(* Logix 5000 project; controller Drives_Line1 1756-L72 rev 20.13; software revision 20.04; part 2 of 21 *)
(* tags used below, declared in another part *)
   TofStitch_Z2 : TIMER;
   TofStitch_Z3 : TIMER;
   TofWatchDogMaster : TIMER;
   _bv_tmp : INT;
   Bridle_01 : UDT_Bridle_3M;
   Bridle_01_FB_Diff : REAL;
   Bridle_01_FB_Update_Valid : BOOL;
   Bridle_01b_FBCounts_mm : REAL;
   Bridle_02 : UDT_Bridle_2M;
   Bridle_03 : UDT_Bridle_2M;
   Bridle_04 : UDT_Bridle_3M;
   cu : UDT_Pinchroll;
   Entry_Accu : UDT_Entry_Accu;
   EntryCmd : UDT_Commands_Zone;
   EntryConfig : UDT_Config_Zone;
   EntryCtrl : UDT_Control_Zone;
   EntryFdbks : UDT_Feedbacks_Zone;
   EntrySetpoints : UDT_Setpoints_Zone;
   EntryStat : UDT_Status_Zone;
   Exit_Accu : UDT_Exit_Accu;
   ExitCtrl : UDT_Control_Zone;
   ExitStat : UDT_Status_Zone;
   In_Commands : UDT_Commands;
   In_Config : UDT_Config;
   In_Setpoints : UDT_Setpoints;
   LineCmd : UDT_Commands_Line;
   LineConfig : UDT_Config_Line;
   LineCtrl : UDT_Control_Line;
   LineFdbks : UDT_Feedbacks_Line;
   LineSetpoints : UDT_Setpoints_Line;
   LineStat : UDT_Status_Line;
   nbrstiychout : DINT;
   Out_Feedbacks : UDT_Fdbks;
   Out_Status : UDT_Status;
   Pinchroll_1 : UDT_Pinchroll;
   Pinchroll_2 : UDT_Pinchroll;
   TestConfig_Line : UDT_Config_Line;
   Unwinder_1 : UDT_Unwinder;
   Unwinder_2 : UDT_Unwinder;
   voirmw : BOOL;
   zConfigFromMaster : BOOL;
   zSimulation : BOOL;
(* P00_Line, continued *)

ROUTINE R12_Line_State   (* ladder *)
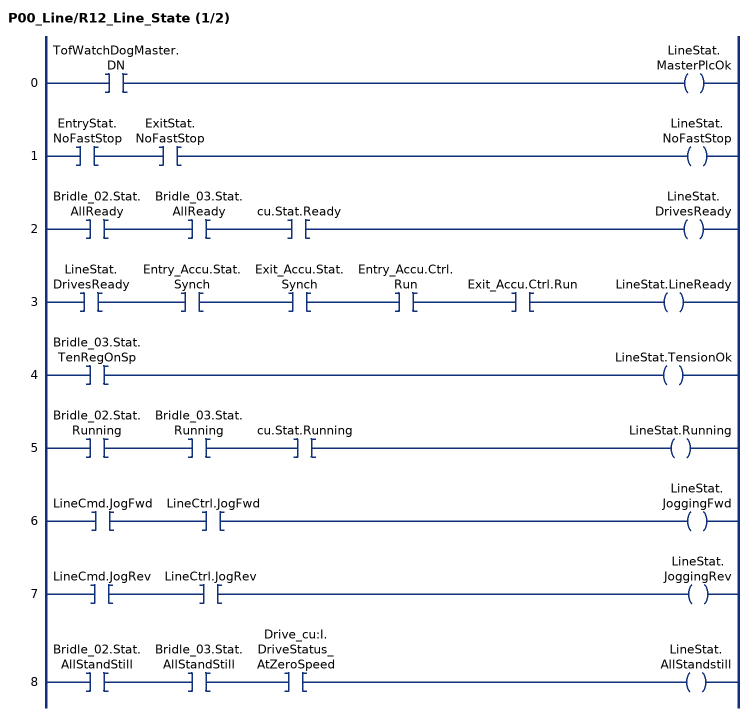
   0: XIC(TofWatchDogMaster.DN)OTE(LineStat.MasterPlcOk);
   1: XIC(EntryStat.NoFastStop)XIC(ExitStat.NoFastStop)OTE(LineStat.NoFastStop);
   2: XIC(Bridle_02.Stat.AllReady)XIC(Bridle_03.Stat.AllReady)XIC(cu.Stat.Ready)OTE(LineStat.DrivesReady);
   3: XIC(LineStat.DrivesReady)XIC(Entry_Accu.Stat.Synch)XIC(Exit_Accu.Stat.Synch)XIC(Entry_Accu.Ctrl.Run)XIC(Exit_Accu.Ctrl.Run)OTE(LineStat.LineReady);
   4: XIC(Bridle_03.Stat.TenRegOnSp)OTE(LineStat.TensionOk);
   5: XIC(Bridle_02.Stat.Running)XIC(Bridle_03.Stat.Running)XIC(cu.Stat.Running)OTE(LineStat.Running);
   6: XIC(LineCmd.JogFwd)XIC(LineCtrl.JogFwd)OTE(LineStat.JoggingFwd);
   7: XIC(LineCmd.JogRev)XIC(LineCtrl.JogRev)OTE(LineStat.JoggingRev);
   8: XIC(Bridle_02.Stat.AllStandStill)XIC(Bridle_03.Stat.AllStandStill)XIC(Drive_cu:I.DriveStatus_AtZeroSpeed)OTE(LineStat.AllStandstill);
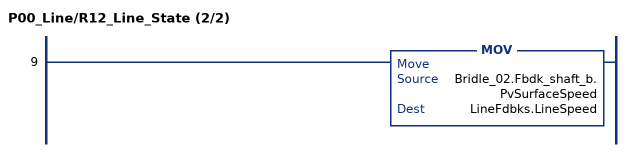
   9: MOV(Bridle_02.Fbdk_shaft_b.PvSurfaceSpeed,LineFdbks.LineSpeed);
END_ROUTINE

ROUTINE R13_Line_Control   (* ladder *)
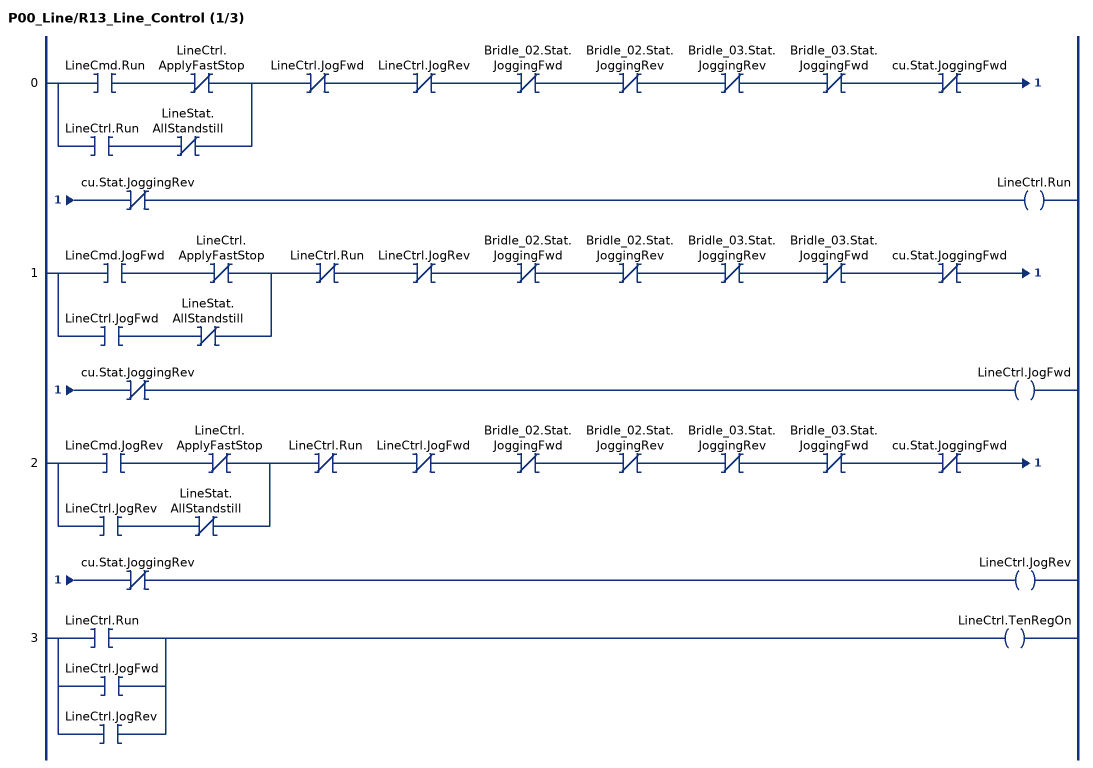
   0: [XIC(LineCmd.Run) XIO(LineCtrl.ApplyFastStop) ,XIC(LineCtrl.Run) XIO(LineStat.AllStandstill) ]XIO(LineCtrl.JogFwd)XIO(LineCtrl.JogRev)XIO(Bridle_02.Stat.JoggingFwd)XIO(Bridle_02.Stat.JoggingRev)XIO(Bridle_03.Stat.JoggingRev)XIO(Bridle_03.Stat.JoggingFwd)XIO(cu.Stat.JoggingFwd)XIO(cu.Stat.JoggingRev)OTE(LineCtrl.Run);
   1: [XIC(LineCmd.JogFwd) XIO(LineCtrl.ApplyFastStop) ,XIC(LineCtrl.JogFwd) XIO(LineStat.AllStandstill) ]XIO(LineCtrl.Run)XIO(LineCtrl.JogRev)XIO(Bridle_02.Stat.JoggingFwd)XIO(Bridle_02.Stat.JoggingRev)XIO(Bridle_03.Stat.JoggingRev)XIO(Bridle_03.Stat.JoggingFwd)XIO(cu.Stat.JoggingFwd)XIO(cu.Stat.JoggingRev)OTE(LineCtrl.JogFwd);
   2: [XIC(LineCmd.JogRev) XIO(LineCtrl.ApplyFastStop) ,XIC(LineCtrl.JogRev) XIO(LineStat.AllStandstill) ]XIO(LineCtrl.Run)XIO(LineCtrl.JogFwd)XIO(Bridle_02.Stat.JoggingFwd)XIO(Bridle_02.Stat.JoggingRev)XIO(Bridle_03.Stat.JoggingRev)XIO(Bridle_03.Stat.JoggingFwd)XIO(cu.Stat.JoggingFwd)XIO(cu.Stat.JoggingRev)OTE(LineCtrl.JogRev);
   3: [XIC(LineCtrl.Run) ,XIC(LineCtrl.JogFwd) ,XIC(LineCtrl.JogRev) ]OTE(LineCtrl.TenRegOn);
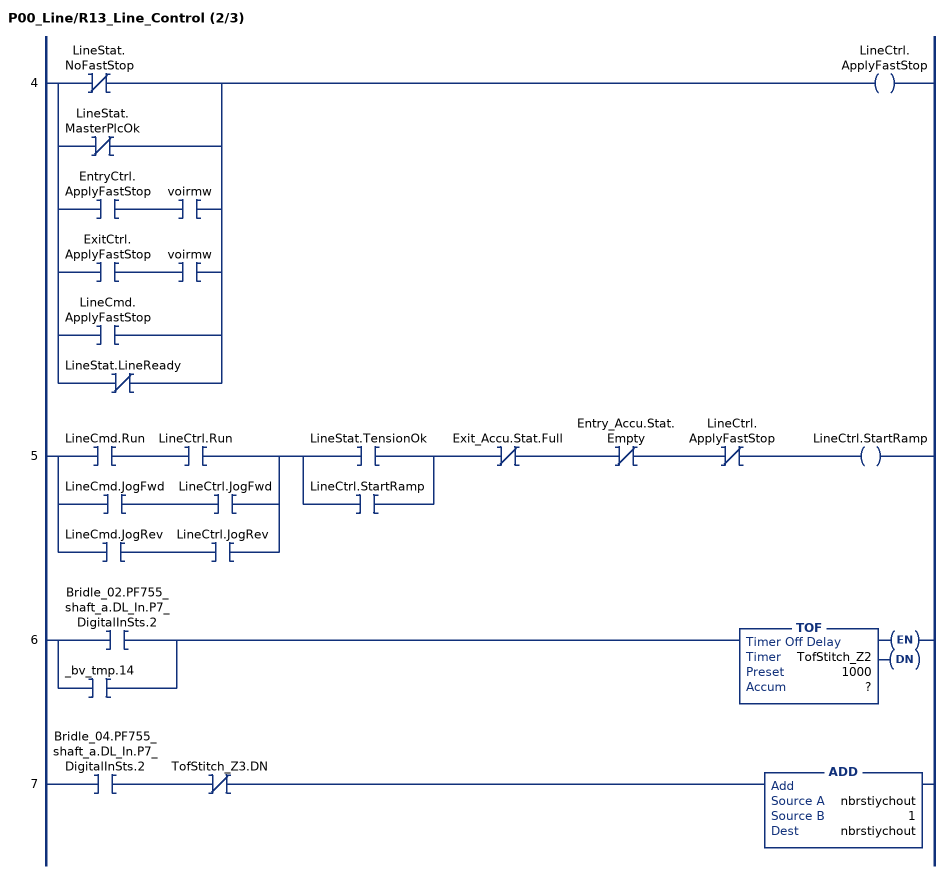
   4: [XIO(LineStat.NoFastStop) ,XIO(LineStat.MasterPlcOk) ,XIC(EntryCtrl.ApplyFastStop) XIC(voirmw) ,XIC(ExitCtrl.ApplyFastStop) XIC(voirmw) ,XIC(LineCmd.ApplyFastStop) ,XIO(LineStat.LineReady) ]OTE(LineCtrl.ApplyFastStop);
   5: [XIC(LineCmd.Run) XIC(LineCtrl.Run) ,XIC(LineCmd.JogFwd) XIC(LineCtrl.JogFwd) ,XIC(LineCmd.JogRev) XIC(LineCtrl.JogRev) ][XIC(LineStat.TensionOk) ,XIC(LineCtrl.StartRamp) ]XIO(Exit_Accu.Stat.Full)XIO(Entry_Accu.Stat.Empty)XIO(LineCtrl.ApplyFastStop)OTE(LineCtrl.StartRamp);
   6: [XIC(Bridle_02.PF755_shaft_a.DL_In.P7_DigitalInSts.2) ,XIC(_bv_tmp.14) ]TOF(TofStitch_Z2,?,?);
   7: XIC(Bridle_04.PF755_shaft_a.DL_In.P7_DigitalInSts.2)XIO(TofStitch_Z3.DN)ADD(nbrstiychout,1,nbrstiychout);
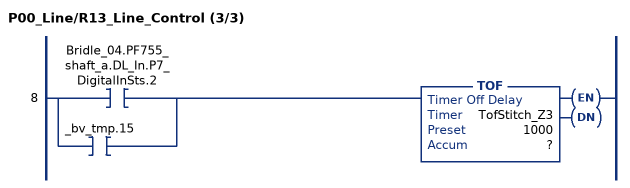
   8: [XIC(Bridle_04.PF755_shaft_a.DL_In.P7_DigitalInSts.2) ,XIC(_bv_tmp.15) ]TOF(TofStitch_Z3,?,?);
END_ROUTINE

ROUTINE R15_Ramp_LineRef_Vp   (* function block diagram *)
   SHEET 1   // Select speed reference
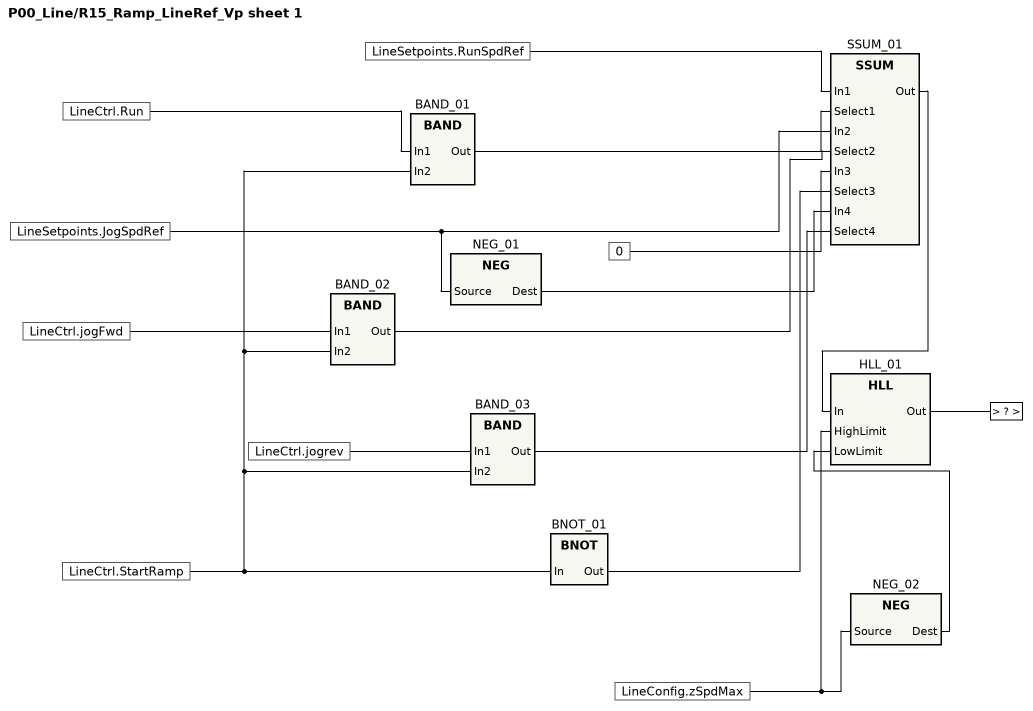
   BAND_02 : BAND(In1 := LineCtrl.jogFwd, In2 := LineCtrl.StartRamp);
   BAND_01 : BAND(In1 := LineCtrl.Run, In2 := LineCtrl.StartRamp);
   NEG_01 : NEG(Source := LineSetpoints.JogSpdRef);
   BAND_03 : BAND(In1 := LineCtrl.jogrev, In2 := LineCtrl.StartRamp);
   BNOT_01 : BNOT(In := LineCtrl.StartRamp);
   SSUM_01 : SSUM(In1 := LineSetpoints.RunSpdRef, Select1 := BAND_01.Out, In2 := LineSetpoints.JogSpdRef, Select2 := BAND_02.Out, In3 := 0, Select3 := BNOT_01.Out, In4 := NEG_01.Dest, Select4 := BAND_03.Out);
   NEG_02 : NEG(Source := LineConfig.zSpdMax);
   HLL_01 : HLL(In := SSUM_01.Out, HighLimit := LineConfig.zSpdMax, LowLimit := NEG_02.Dest);
   WIRE(?) := HLL_01.Out;
   SHEET 2   // Select acceleration rate
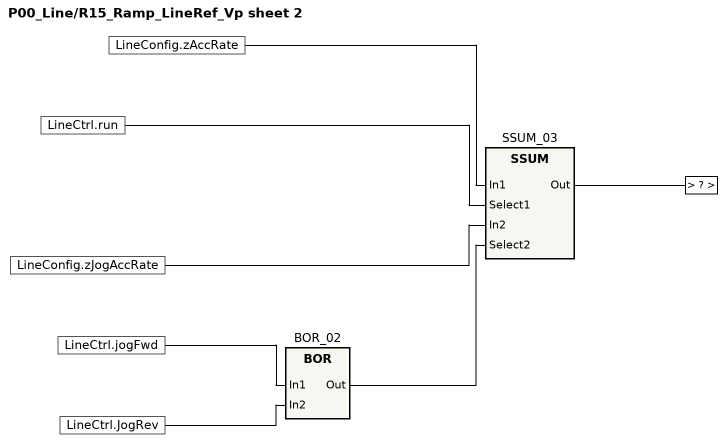
   BOR_02 : BOR(In1 := LineCtrl.jogFwd, In2 := LineCtrl.JogRev);
   SSUM_03 : SSUM(In1 := LineConfig.zAccRate, Select1 := LineCtrl.run, In2 := LineConfig.zJogAccRate, Select2 := BOR_02.Out);
   WIRE(?) := SSUM_03.Out;
   SHEET 3   // Select deceleration rate
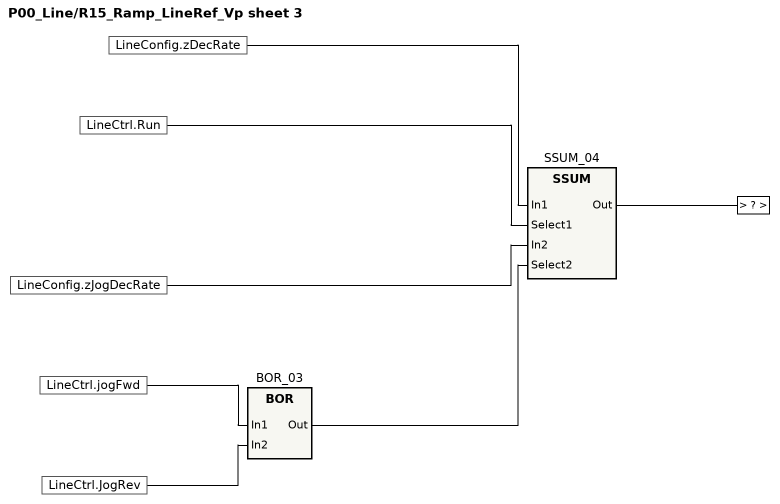
   BOR_03 : BOR(In1 := LineCtrl.jogFwd, In2 := LineCtrl.JogRev);
   SSUM_04 : SSUM(In1 := LineConfig.zDecRate, Select1 := LineCtrl.Run, In2 := LineConfig.zJogDecRate, Select2 := BOR_03.Out);
   WIRE(?) := SSUM_04.Out;
   SHEET 4   // S-Curve line speed (Vp)
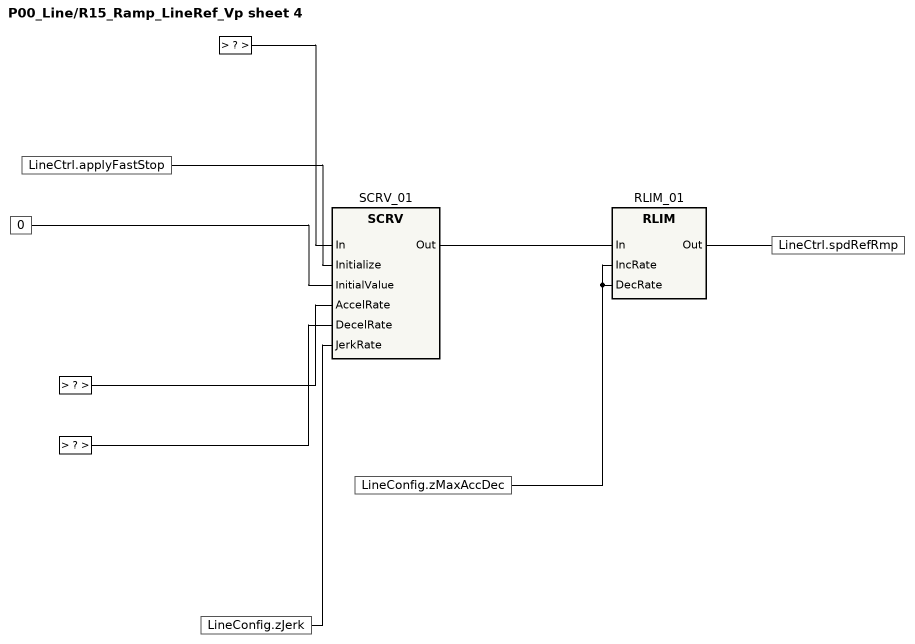
   SCRV_01 : SCRV(In := WIRE(?), Initialize := LineCtrl.applyFastStop, InitialValue := 0, AccelRate := WIRE(?), DecelRate := WIRE(?), JerkRate := LineConfig.zJerk);
   RLIM_01 : RLIM(In := SCRV_01.Out, IncRate := LineConfig.zMaxAccDec, DecRate := LineConfig.zMaxAccDec);
   LineCtrl.spdRefRmp := RLIM_01.Out;
END_ROUTINE

ROUTINE R999_Test   (* ladder *)
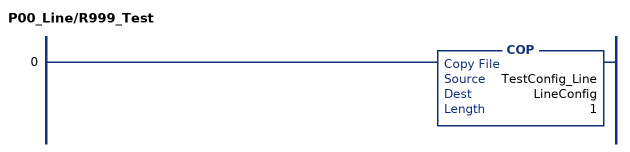
   0: COP(TestConfig_Line,LineConfig,1);
END_ROUTINE

ROUTINE R99_To_Master   (* ladder *)
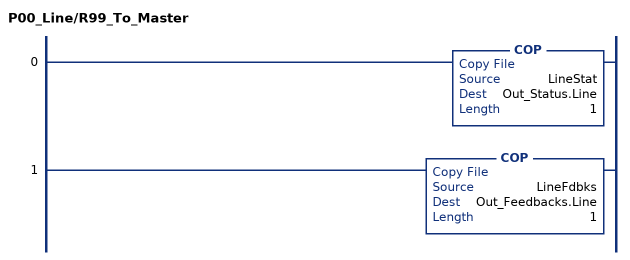
   0: COP(LineStat,Out_Status.Line,1);
   1: COP(LineFdbks,Out_Feedbacks.Line,1);
END_ROUTINE
END_PROGRAM

PROGRAM P01_Entry_Zone   (* main routine R00_Main *)
VAR
   BAND_10 : FBD_BOOLEAN_AND := (In3 := 1, In4 := 1, In5 := 1, In6 := 1, In7 := 1, In8 := 1);
   BAND_11 : FBD_BOOLEAN_AND := (In3 := 1, In4 := 1, In5 := 1, In6 := 1, In7 := 1, In8 := 1);
   BAND_12 : FBD_BOOLEAN_AND := (In3 := 1, In4 := 1, In5 := 1, In6 := 1, In7 := 1, In8 := 1);
   BNOT_01 : FBD_BOOLEAN_NOT := (Out := 1);
   BNOT_04 : FBD_BOOLEAN_NOT := (Out := 1);
   BOR_01 : FBD_BOOLEAN_OR;
   Entry_PosPv_Shear_Stitch : REAL := 2345.455;
   Entry_PosPv_Stitch_HOC : DINT;
   Entry_PosSp_AtShear : DINT := 1650;
   Entry_PosSp_AtStitch_EOC : DINT := 2345;
   Entry_PosSp_AtStitch_HOC : DINT := 1650;
   EOC_PosStitchStep : DINT;
   EOC_ToShearStep : DINT;
   HLL_01 : HL_LIMIT := (HighLimit := 0.5, LowLimit := -0.5);
   HLL_02 : HL_LIMIT := (HighAlarm := 1, LowAlarm := 1, Status := 16#0000_0003, InstructFault := 1, LimitsInv := 1);
   HOC_ToStitchStep : DINT;
   NEG_01 : FBD_MATH_ADVANCED := (Source := 0.5, Dest := -0.5);
   NEG_05 : FBD_MATH_ADVANCED := (Source := 0.1, Dest := -0.1);
   NEG_06 : FBD_MATH_ADVANCED;
   ons : BOOL[32] := ([0] := 1, [1] := 1);
   RLIM_02 : RATE_LIMITER := (IncRate := 0.25, DecRate := 0.25, RTSTime := 1, DeltaT := 0.05);
   SCRV_02 : S_CURVE := (Initialize := 1, RTSTime := 1, DeltaT := 0.05);
   SEL_02 : SELECT := (In1 := 0.08, SelectorIn := 1);
   SSUM_03 : SELECTED_SUMMER := (Gain1 := 1.0, In2 := 0.1, Gain2 := 1.0, In3 := -0.1, Gain3 := 1.0, Gain4 := 1.0, Select4 := 1, Gain5 := 1.0, Gain6 := 1.0, Gain7 := 1.0, Gain8 := 1.0);
   SSUM_06 : SELECTED_SUMMER := (In1 := 0.04, Gain1 := 1.0, In2 := 0.083, Gain2 := 1.0, Gain3 := 1.0, Gain4 := 1.0, Gain5 := 1.0, Gain6 := 1.0, Gain7 := 1.0, Gain8 := 1.0);
   SSUM_08 : SELECTED_SUMMER := (In1 := 0.04, Gain1 := 1.0, In2 := 0.083, Gain2 := 1.0, Gain3 := 1.0, Gain4 := 1.0, Gain5 := 1.0, Gain6 := 1.0, Gain7 := 1.0, Gain8 := 1.0);
   SSUM_09 : SELECTED_SUMMER := (In1 := 0.15, Gain1 := 1.0, In2 := 0.1, Gain2 := 1.0, Gain3 := 1.0, Gain4 := 1.0, Gain5 := 1.0, Gain6 := 1.0, Gain7 := 1.0, Gain8 := 1.0);
   Ton_EOC_Sensor : TIMER := (PRE := 1000, ACC := 1000, EN := 1, DN := 1);
   TonRefOn : TIMER := (PRE := 750);
   zEntry_Dist_Pinch_Shear : REAL := 1650.0;
   zEntry_Dist_ShearToStitch : REAL := 695.0;
   zMaxSpdEntryNotSync : REAL := 0.08;
END_VAR

ROUTINE R00_Main   (* ladder *)
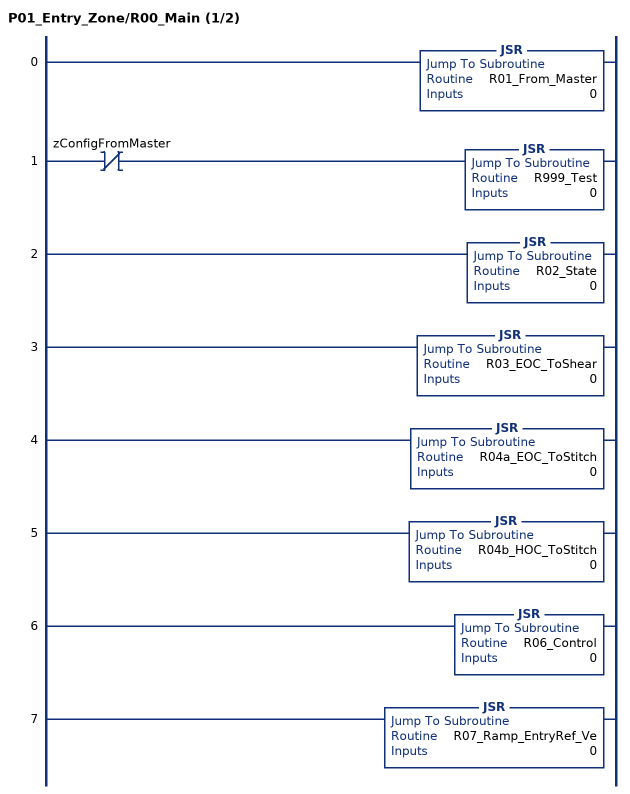
   0: JSR(R01_From_Master,0);
   1: XIO(zConfigFromMaster)JSR(R999_Test,0);
   2: JSR(R02_State,0);
   3: JSR(R03_EOC_ToShear,0);
   4: JSR(R04a_EOC_ToStitch,0);
   5: JSR(R04b_HOC_ToStitch,0);
   6: JSR(R06_Control,0);
   7: JSR(R07_Ramp_EntryRef_Ve,0);
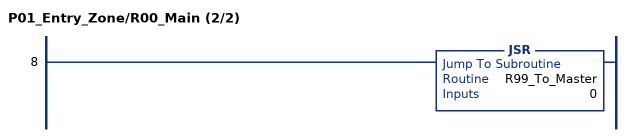
   8: JSR(R99_To_Master,0);
END_ROUTINE

ROUTINE R01_From_Master   (* ladder *)
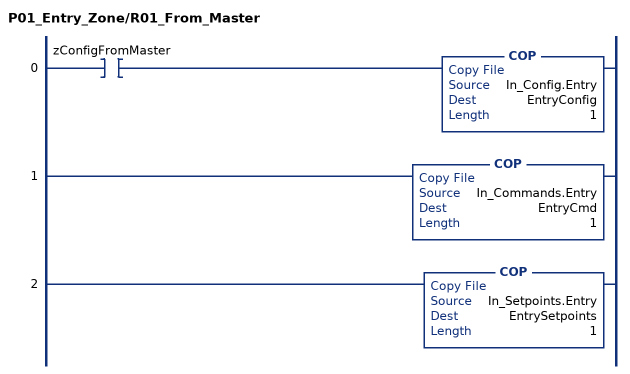
   0: XIC(zConfigFromMaster)COP(In_Config.Entry,EntryConfig,1);
   1: COP(In_Commands.Entry,EntryCmd,1);
   2: COP(In_Setpoints.Entry,EntrySetpoints,1);
END_ROUTINE

ROUTINE R02_State   (* ladder *)
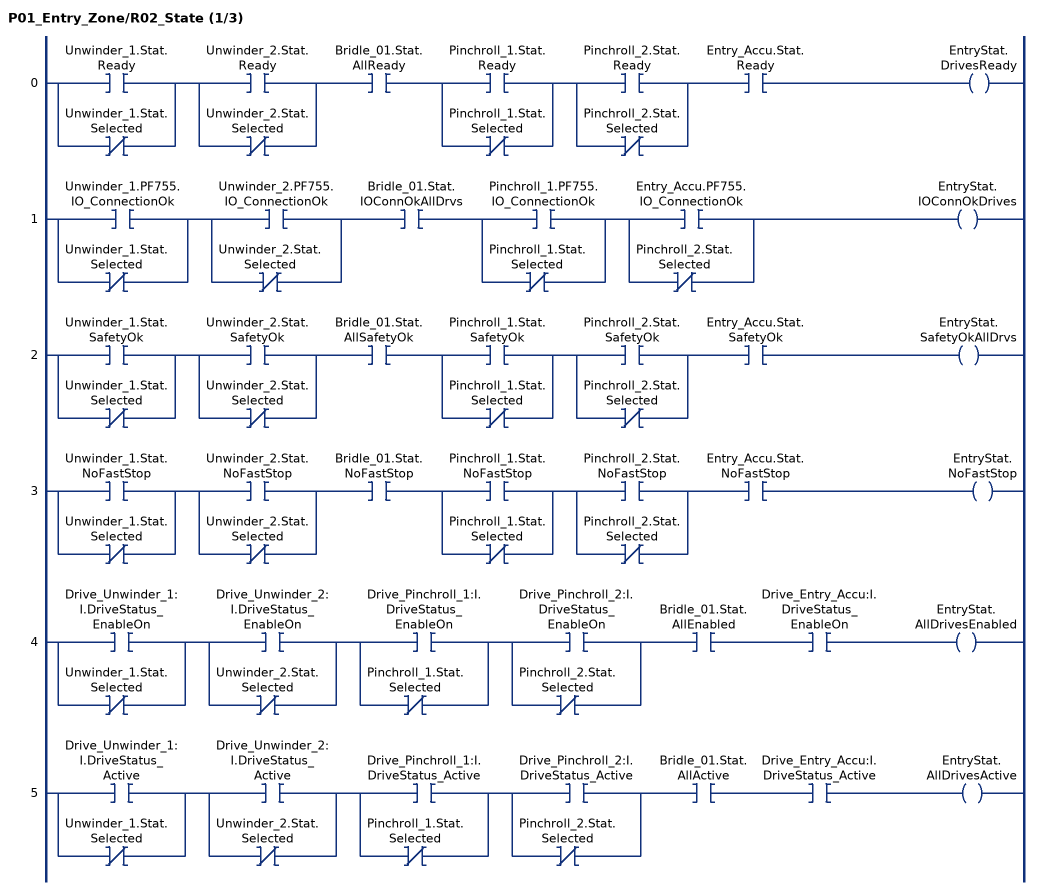
   0: [XIC(Unwinder_1.Stat.Ready) ,XIO(Unwinder_1.Stat.Selected) ][XIC(Unwinder_2.Stat.Ready) ,XIO(Unwinder_2.Stat.Selected) ]XIC(Bridle_01.Stat.AllReady)[XIC(Pinchroll_1.Stat.Ready) ,XIO(Pinchroll_1.Stat.Selected) ][XIC(Pinchroll_2.Stat.Ready) ,XIO(Pinchroll_2.Stat.Selected) ]XIC(Entry_Accu.Stat.Ready)OTE(EntryStat.DrivesReady);
   1: [XIC(Unwinder_1.PF755.IO_ConnectionOk) ,XIO(Unwinder_1.Stat.Selected) ][XIC(Unwinder_2.PF755.IO_ConnectionOk) ,XIO(Unwinder_2.Stat.Selected) ]XIC(Bridle_01.Stat.IOConnOkAllDrvs)[XIC(Pinchroll_1.PF755.IO_ConnectionOk) ,XIO(Pinchroll_1.Stat.Selected) ][XIC(Entry_Accu.PF755.IO_ConnectionOk) ,XIO(Pinchroll_2.Stat.Selected) ]OTE(EntryStat.IOConnOkDrives);
   2: [XIC(Unwinder_1.Stat.SafetyOk) ,XIO(Unwinder_1.Stat.Selected) ][XIC(Unwinder_2.Stat.SafetyOk) ,XIO(Unwinder_2.Stat.Selected) ]XIC(Bridle_01.Stat.AllSafetyOk)[XIC(Pinchroll_1.Stat.SafetyOk) ,XIO(Pinchroll_1.Stat.Selected) ][XIC(Pinchroll_2.Stat.SafetyOk) ,XIO(Pinchroll_2.Stat.Selected) ]XIC(Entry_Accu.Stat.SafetyOk)OTE(EntryStat.SafetyOkAllDrvs);
   3: [XIC(Unwinder_1.Stat.NoFastStop) ,XIO(Unwinder_1.Stat.Selected) ][XIC(Unwinder_2.Stat.NoFastStop) ,XIO(Unwinder_2.Stat.Selected) ]XIC(Bridle_01.Stat.NoFastStop)[XIC(Pinchroll_1.Stat.NoFastStop) ,XIO(Pinchroll_1.Stat.Selected) ][XIC(Pinchroll_2.Stat.NoFastStop) ,XIO(Pinchroll_2.Stat.Selected) ]XIC(Entry_Accu.Stat.NoFastStop)OTE(EntryStat.NoFastStop);
   4: [XIC(Drive_Unwinder_1:I.DriveStatus_EnableOn) ,XIO(Unwinder_1.Stat.Selected) ][XIC(Drive_Unwinder_2:I.DriveStatus_EnableOn) ,XIO(Unwinder_2.Stat.Selected) ][XIC(Drive_Pinchroll_1:I.DriveStatus_EnableOn) ,XIO(Pinchroll_1.Stat.Selected) ][XIC(Drive_Pinchroll_2:I.DriveStatus_EnableOn) ,XIO(Pinchroll_2.Stat.Selected) ]XIC(Bridle_01.Stat.AllEnabled)XIC(Drive_Entry_Accu:I.DriveStatus_EnableOn)OTE(EntryStat.AllDrivesEnabled);
   5: [XIC(Drive_Unwinder_1:I.DriveStatus_Active) ,XIO(Unwinder_1.Stat.Selected) ][XIC(Drive_Unwinder_2:I.DriveStatus_Active) ,XIO(Unwinder_2.Stat.Selected) ][XIC(Drive_Pinchroll_1:I.DriveStatus_Active) ,XIO(Pinchroll_1.Stat.Selected) ][XIC(Drive_Pinchroll_2:I.DriveStatus_Active) ,XIO(Pinchroll_2.Stat.Selected) ]XIC(Bridle_01.Stat.AllActive)XIC(Drive_Entry_Accu:I.DriveStatus_Active)OTE(EntryStat.AllDrivesActive);
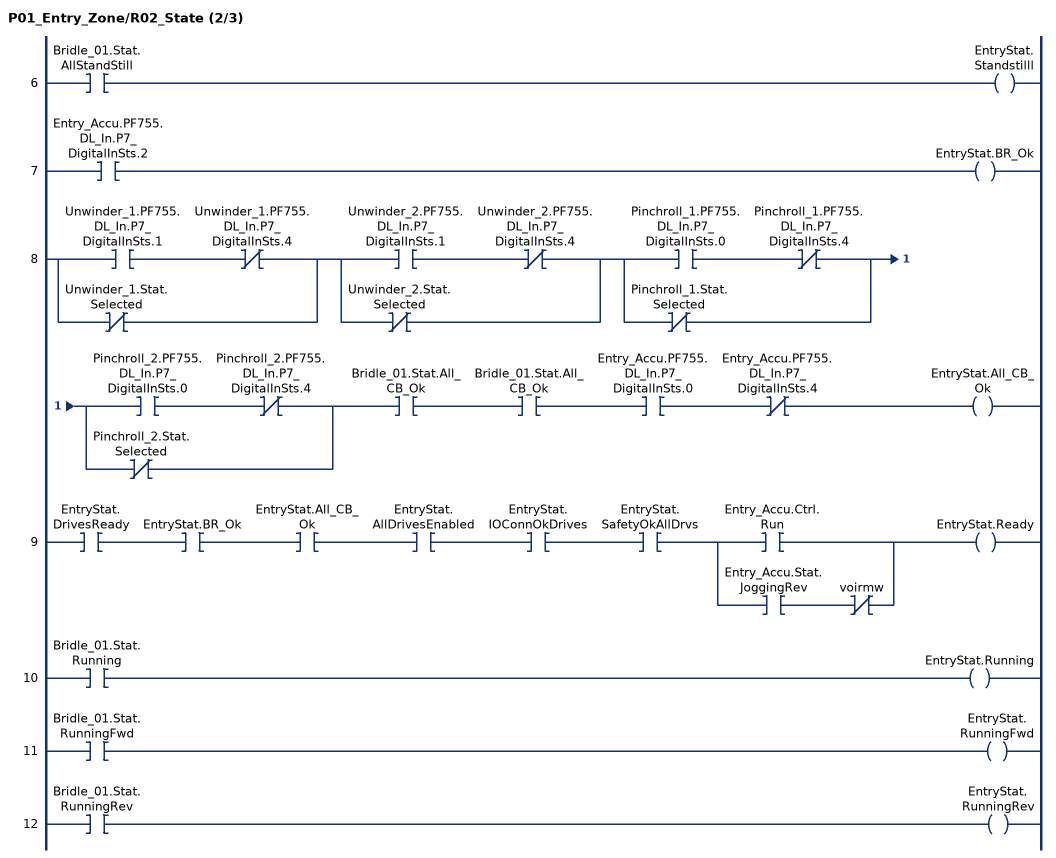
   6: XIC(Bridle_01.Stat.AllStandStill)OTE(EntryStat.Standstilll);
   7: XIC(Entry_Accu.PF755.DL_In.P7_DigitalInSts.2)OTE(EntryStat.BR_Ok);
   8: [XIC(Unwinder_1.PF755.DL_In.P7_DigitalInSts.1) XIO(Unwinder_1.PF755.DL_In.P7_DigitalInSts.4) ,XIO(Unwinder_1.Stat.Selected) ][XIC(Unwinder_2.PF755.DL_In.P7_DigitalInSts.1) XIO(Unwinder_2.PF755.DL_In.P7_DigitalInSts.4) ,XIO(Unwinder_2.Stat.Selected) ][XIC(Pinchroll_1.PF755.DL_In.P7_DigitalInSts.0) XIO(Pinchroll_1.PF755.DL_In.P7_DigitalInSts.4) ,XIO(Pinchroll_1.Stat.Selected) ][XIC(Pinchroll_2.PF755.DL_In.P7_DigitalInSts.0) XIO(Pinchroll_2.PF755.DL_In.P7_DigitalInSts.4) ,XIO(Pinchroll_2.Stat.Selected) ]XIC(Bridle_01.Stat.All_CB_Ok)XIC(Bridle_01.Stat.All_CB_Ok)XIC(Entry_Accu.PF755.DL_In.P7_DigitalInSts.0)XIO(Entry_Accu.PF755.DL_In.P7_DigitalInSts.4)OTE(EntryStat.All_CB_Ok);
   9: XIC(EntryStat.DrivesReady)XIC(EntryStat.BR_Ok)XIC(EntryStat.All_CB_Ok)XIC(EntryStat.AllDrivesEnabled)XIC(EntryStat.IOConnOkDrives)XIC(EntryStat.SafetyOkAllDrvs)[XIC(Entry_Accu.Ctrl.Run) ,XIC(Entry_Accu.Stat.JoggingRev) XIO(voirmw) ]OTE(EntryStat.Ready);
   10: XIC(Bridle_01.Stat.Running)OTE(EntryStat.Running);
   11: XIC(Bridle_01.Stat.RunningFwd)OTE(EntryStat.RunningFwd);
   12: XIC(Bridle_01.Stat.RunningRev)OTE(EntryStat.RunningRev);
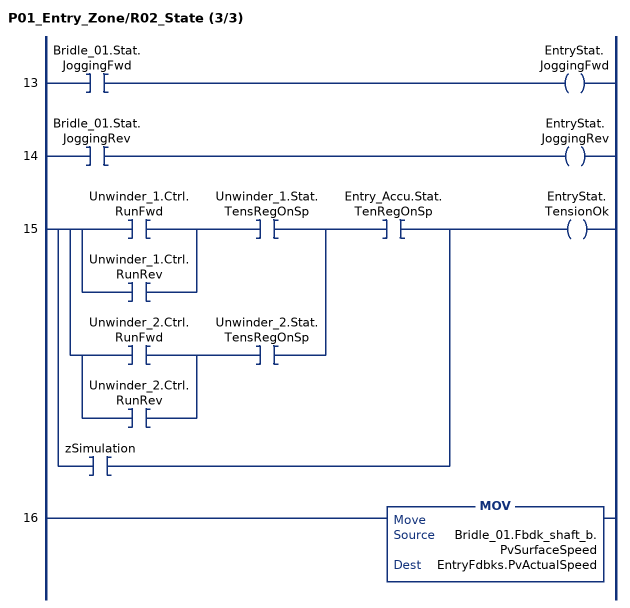
   13: XIC(Bridle_01.Stat.JoggingFwd)OTE(EntryStat.JoggingFwd);
   14: XIC(Bridle_01.Stat.JoggingRev)OTE(EntryStat.JoggingRev);
   15: [[[XIC(Unwinder_1.Ctrl.RunFwd) ,XIC(Unwinder_1.Ctrl.RunRev) ] XIC(Unwinder_1.Stat.TensRegOnSp) ,[XIC(Unwinder_2.Ctrl.RunFwd) ,XIC(Unwinder_2.Ctrl.RunRev) ] XIC(Unwinder_2.Stat.TensRegOnSp) ] XIC(Entry_Accu.Stat.TenRegOnSp) ,XIC(zSimulation) ]OTE(EntryStat.TensionOk);
   16: MOV(Bridle_01.Fbdk_shaft_b.PvSurfaceSpeed,EntryFdbks.PvActualSpeed);
END_ROUTINE

ROUTINE R03_EOC_ToShear   (* ladder *)
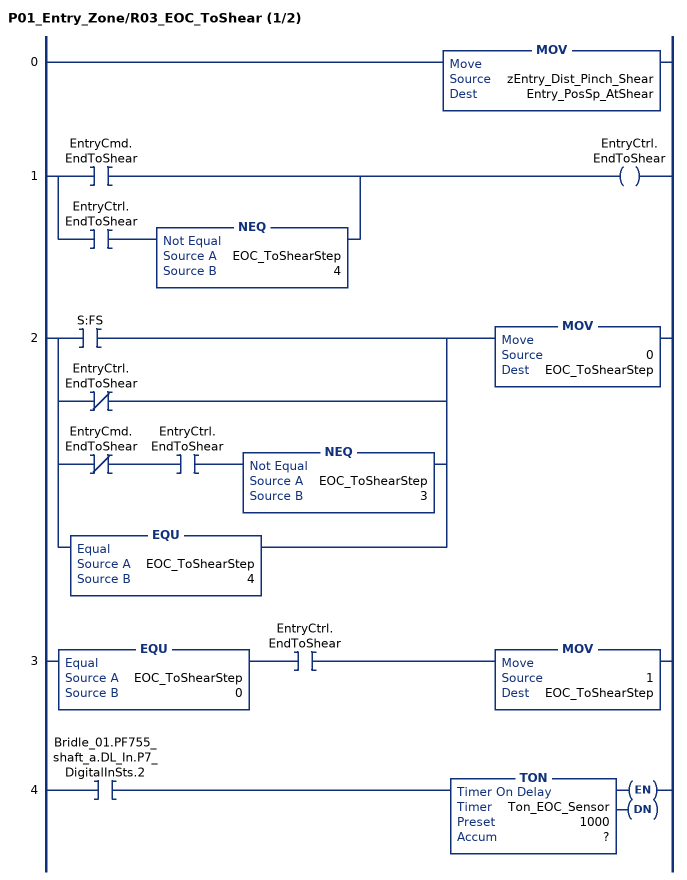
   0: MOV(zEntry_Dist_Pinch_Shear,Entry_PosSp_AtShear);
   1: [XIC(EntryCmd.EndToShear) ,XIC(EntryCtrl.EndToShear) NEQ(EOC_ToShearStep,4) ]OTE(EntryCtrl.EndToShear);
   2: [XIC(S:FS) ,XIO(EntryCtrl.EndToShear) ,XIO(EntryCmd.EndToShear) XIC(EntryCtrl.EndToShear) NEQ(EOC_ToShearStep,3) ,EQU(EOC_ToShearStep,4) ]MOV(0,EOC_ToShearStep);
   3: EQU(EOC_ToShearStep,0)XIC(EntryCtrl.EndToShear)MOV(1,EOC_ToShearStep);
   4: XIC(Bridle_01.PF755_shaft_a.DL_In.P7_DigitalInSts.2)TON(Ton_EOC_Sensor,?,?);
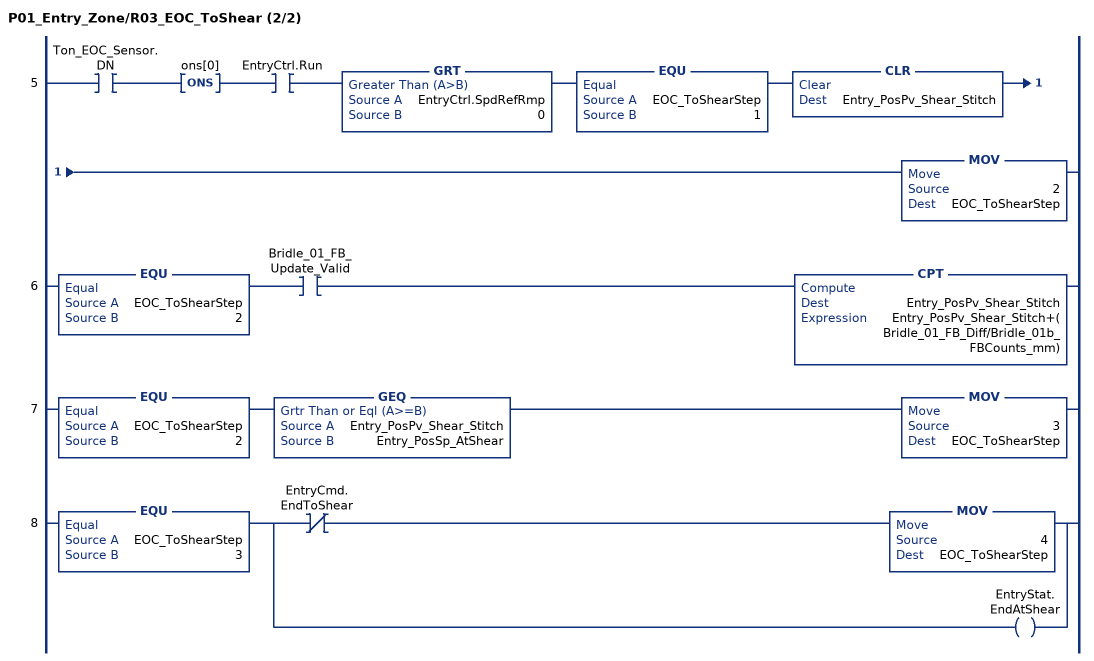
   5: XIC(Ton_EOC_Sensor.DN)ONS(ons[0])XIC(EntryCtrl.Run)GRT(EntryCtrl.SpdRefRmp,0)EQU(EOC_ToShearStep,1)CLR(Entry_PosPv_Shear_Stitch)MOV(2,EOC_ToShearStep);
   6: EQU(EOC_ToShearStep,2)XIC(Bridle_01_FB_Update_Valid)CPT(Entry_PosPv_Shear_Stitch,Entry_PosPv_Shear_Stitch+(Bridle_01_FB_Diff/Bridle_01b_FBCounts_mm));
   7: EQU(EOC_ToShearStep,2)GEQ(Entry_PosPv_Shear_Stitch,Entry_PosSp_AtShear)MOV(3,EOC_ToShearStep);
   8: EQU(EOC_ToShearStep,3)[XIO(EntryCmd.EndToShear) MOV(4,EOC_ToShearStep) ,OTE(EntryStat.EndAtShear) ];
END_ROUTINE
